(* PLC project  *)

CONFIGURATION EL1904
END_CONFIGURATION
